// TwinCAT 3 PLC project Blinker
// ProgramVersion: 3.1.4024.0
// libraries:
//   Tc2_Standard, * (Beckhoff Automation GmbH)
//   Tc2_System, * (Beckhoff Automation GmbH)
//   Tc3_Module, * (Beckhoff Automation GmbH)
//   VisuDialogs, * (System)
// project tree:
//   DUTs/ E_BlinkerPhase.TcDUT
//   / GlobalTextList.TcGTLO, PlcTask.TcTTO, Visualization Manager.TcVMO (not stored)
//   POUs/ FB_Blinker.TcPOU, FB_CaseBlinker.TcPOU, MAIN.TcPOU
//   VISUs/ Visualization.TcVIS
// real-time tasks:
//   TASK PlcTask: cycle T#10ms, priority 20, ADS port 350
// I/O:
//   DEVICE Device 2 (EtherCAT) (disabled), AmsNetId 10.0.20.81.3.1
//     Term 1 (EK1100) [EK1100 EtherCAT Coupler (2A E-Bus)]
//       Term 2 (EL1014) [EL1014 4Ch. Dig. Input 24V, 10µs]
//       Term 3 (EL2004) [EL2004 4Ch. Dig. Output 24V, 0.5A]
//       Term 4 (EL9011) [EL9011 End Terminal]
// variable links:
//   Blinker/Blinker Instance <-> Device 2 (EtherCAT)/Term 1 (EK1100)/Term 2 (EL1014)
//     PlcTask Inputs/MAIN.fbCaseBlinker.bIsStartPressed <-> Channel 1/Input
//   Blinker/Blinker Instance <-> Device 2 (EtherCAT)/Term 1 (EK1100)/Term 3 (EL2004)
//     PlcTask Outputs/MAIN.fbCaseBlinker.bLight <-> Channel 1/Output

CONFIGURATION Blinker
    RESOURCE PLC ON TwinCAT3
        TASK PlcTask(INTERVAL := T#10ms, PRIORITY := 20);
        PROGRAM MAIN WITH PlcTask : MAIN;
    END_RESOURCE
END_CONFIGURATION

// ---- DUTs/E_BlinkerPhase.TcDUT
{attribute 'qualified_only'}
{attribute 'strict'}
TYPE E_BlinkerPhase :
(
	IdlePhase := 0,
	OnPhase := 10,
	OffPhase := 20
);
END_TYPE

// ---- POUs/MAIN.TcPOU
PROGRAM MAIN
VAR
	fbBlinker : FB_Blinker;
	fbCaseBlinker : FB_CaseBlinker;
	
	bIsStartPressed : BOOL;
	bIsCaseStartPressed : BOOL;
	
	dwTimeOn : DWORD := 2000;
	dwTimeOff : DWORD := 1000;
	dwCaseTimeOn : DWORD := 2000;
	dwCaseTimeOff : DWORD := 1000;
END_VAR

fbBlinker(bIsStartPressed := bIsStartPressed, dwTimeOn := dwTimeOn, dwTimeOff := dwTimeOff);

fbCaseBlinker(bIsStartPressed := bIsCaseStartPressed, dwTimeOn := dwCaseTimeOn, dwTimeOff := dwCaseTimeOff);

fbCaseBlinker(dwTimeOn := dwCaseTimeOn, dwTimeOff := dwCaseTimeOff);

END_PROGRAM

// ---- POUs/FB_Blinker.TcPOU
FUNCTION_BLOCK FB_Blinker
VAR_INPUT
	bIsStartPressed : BOOL;
	dwTimeOn : DWORD;
	dwTimeOff : DWORD;
END_VAR
VAR_OUTPUT
	bLight : BOOL;	// Determines whether the light will be ON or OFF
END_VAR
VAR
	fbTimerOn : TON;
	fbTimerOff : TON;
	fbStartTrigger : R_TRIG;
	
	bCurrentPhase : BOOL;	// Tracks whether we are in the ON phase or OFF phase
	bIsBlinking : bool;
END_VAR

// Detect whether the start button is pressed
fbStartTrigger(CLK := bIsStartPressed);
IF fbStartTrigger.Q THEN
    bIsBlinking := NOT bIsBlinking; // Toggle the blinking state (start or stop blinking)
END_IF

IF bIsBlinking THEN
    IF bCurrentPhase THEN
        // Start the on timer
        fbTimerOn(IN := TRUE, PT := DWORD_TO_TIME(dwTimeOn));
        IF fbTimerOn.Q THEN
            bCurrentPhase := FALSE;
            fbTimerOn(IN := FALSE); // Reset the on timer
        END_IF
        bLight := TRUE;
    ELSE
        // Start the off timer
        fbTimerOff(IN := TRUE, PT := DWORD_TO_TIME(dwTimeOff));
        IF fbTimerOff.Q THEN
            bCurrentPhase := TRUE;
            fbTimerOff(IN := FALSE); // Reset the off timer
        END_IF
        bLight := FALSE;
    END_IF
ELSE
    // Reset timers and light when blinking is not active
    fbTimerOn(IN := FALSE);
    fbTimerOff(IN := FALSE);
    bLight := FALSE;
    bCurrentPhase := TRUE;
END_IF

END_FUNCTION_BLOCK

// ---- POUs/FB_CaseBlinker.TcPOU
FUNCTION_BLOCK FB_CaseBlinker
VAR_INPUT
	bIsStartPressed AT %I* : BOOL;
	dwTimeOn : DWORD;
	dwTimeOff : DWORD;
END_VAR
VAR_OUTPUT
	bLight AT %Q* : BOOL;	// Determines whether the light will be ON or OFF
END_VAR
VAR
	fbTimerOn : TON;
	fbTimerOff : TON;
	fbStartTrigger : R_TRIG;
	
	eCurrentPhase : E_BlinkerPhase := 0;	// 0 - Idle, 10 - ON, 20 - OFF
	
	bIsBlinking : bool;
END_VAR

// This blinker is solved using the CASE instruction

// Detect whether the start button is pressed
fbStartTrigger(CLK := bIsStartPressed);
IF fbStartTrigger.Q THEN
    bIsBlinking := NOT bIsBlinking; // Toggle the blinking state (start or stop blinking)
	IF bIsBlinking THEN
		eCurrentPhase := 10;
	ELSE
		eCurrentPhase := 0;
	END_IF
END_IF

CASE eCurrentPhase OF
    0:
        fbTimerOn(IN := FALSE);
        fbTimerOff(IN := FALSE);
        bLight := FALSE;

    10:
        fbTimerOn(IN := TRUE, PT := DWORD_TO_TIME(dwTimeOn));
        IF fbTimerOn.Q THEN
            fbTimerOn(IN := FALSE); // Reset the on timer
            eCurrentPhase := 20;  // Move to the off phase
        END_IF
        bLight := TRUE;

    20:
        fbTimerOff(IN := TRUE, PT := DWORD_TO_TIME(dwTimeOff));
        IF fbTimerOff.Q THEN
            fbTimerOff(IN := FALSE); // Reset the off timer
            eCurrentPhase := 10;  // Move to the On phase
        END_IF
        bLight := FALSE;
END_CASE

END_FUNCTION_BLOCK

// ---- GlobalTextList.TcGTLO
TEXTLIST GlobalTextList
  606 = 'Change light OFF time'
  907 = 'Change light ON time'
  292 = 'Elapsed time: %s'
  452 = 'Light off time'
  757 = 'Light on time'
  362 = 'Solved using CASE:'
  419 = 'START'
  747 = 'START / STOP'
END_TEXTLIST

// ---- VISUs/Visualization.TcVIS
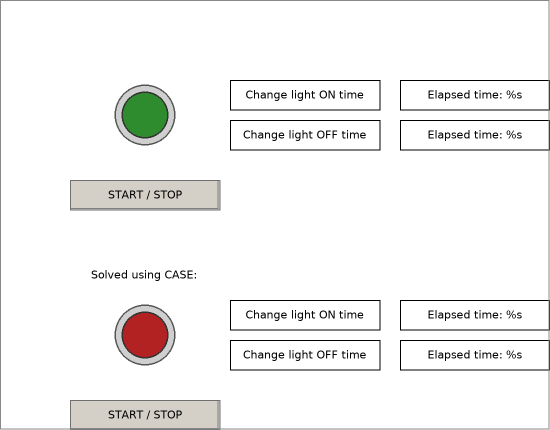
VISUALIZATION Visualization  // 550x430
    Lamp1 (110,80 70x70), variable: MAIN.fbBlinker.bLight, style: Lamp-Lamp1-Green
    Rectangle (230,80 150x30), "Change light ON time"
        OnMouseClick: write MAIN.dwTimeOn via Default
    Rectangle (230,120 150x30), "Change light OFF time"
        OnMouseClick: write MAIN.dwTimeOff via Default
    Button (70,180 150x30), "START / STOP"
        tap MAIN.bIsStartPressed
    Rectangle (400,80 150x30), "Elapsed time: %s", text variable: MAIN.fbBlinker.fbTimerOn.ET
    Rectangle (400,120 150x30), "Elapsed time: %s", text variable: MAIN.fbBlinker.fbTimerOff.ET
    Lamp1 (110,300 70x70), variable: MAIN.fbCaseBlinker.bLight, style: Lamp-Lamp1-Red
    Rectangle (230,300 150x30), "Change light ON time"
        OnMouseClick: write MAIN.dwCaseTimeOn via Default
    Rectangle (230,340 150x30), "Change light OFF time"
        OnMouseClick: write MAIN.dwCaseTimeOff via Default
    Button (70,400 150x30), "START / STOP"
        tap MAIN.bIsCaseStartPressed
    Rectangle (400,340 150x30), "Elapsed time: %s", text variable: MAIN.fbCaseBlinker.fbTimerOff.ET
    Rectangle (400,300 150x30), "Elapsed time: %s", text variable: MAIN.fbCaseBlinker.fbTimerOn.ET
    Rectangle (69,260 150x30), "Solved using CASE:"
END_VISUALIZATION
